FUNCTION_BLOCK IF_VALOR_REAL (* Basic Function Block Type *)
  (* Standard: 61499-2 *)
  (* Version 0.0, 1/23/2026, Schneider Electric, Template *)
  PACKAGE Hidryco.HidrycoLib;
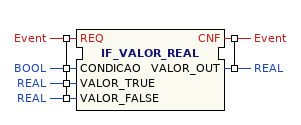
  EVENT_INPUT
    REQ WITH CONDICAO, VALOR_TRUE, VALOR_FALSE; (* Normal Execution Request *)
  END_EVENT
  EVENT_OUTPUT
    CNF WITH VALOR_OUT; (* Execution Confirmation *)
  END_EVENT
  VAR_INPUT
    CONDICAO : BOOL; (* Input event qualifier *)
    VALOR_TRUE : REAL;
    VALOR_FALSE : REAL;
  END_VAR
  VAR_OUTPUT
    VALOR_OUT : REAL;
  END_VAR
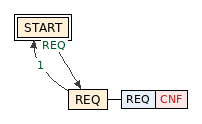
  EC_STATES
    START; (* Initial State *)
    REQ : REQ -> CNF; (* Normal execution *)
  END_STATES
  EC_TRANSITIONS
    START TO REQ := REQ;
    REQ TO START := 1;
  END_TRANSITIONS
  ALGORITHM INIT IN ST: (* Initialization algorithm *)
;
  END_ALGORITHM
  ALGORITHM REQ IN ST: (* Normally executed algorithm *)
IF (CONDICAO) THEN
	VALOR_OUT := VALOR_TRUE;
ELSE
	VALOR_OUT := VALOR_FALSE;
END_IF
;
  END_ALGORITHM
END_FUNCTION_BLOCK
